FUNCTION_BLOCK F_IS_VALID (* Check if REAL/LREAL is valid (not NaN, not Inf) *)
  (* Standard: 61131-3; Description: Copyright (c) 2013 TU Wien ACIN and others. This program and the accompanying materials are made available under the terms of the Eclipse Public License 2.0 which is available at https://www.eclipse.org/legal/epl-2.0/ SPDX-License-Identifier: EPL-2.0 Some portions generated by Gemini CLI *)
  (* Version 3.1, 2026-01-31, Franz Höpfinger, HR Agrartechnik GmbH, initial API and implementation and/or initial documentation *)
  (* Version 3.0, 2025-04-14, Patrick Aigner, changed package *)
  PACKAGE iec61131::conversion;
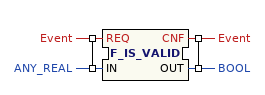
  EVENT_INPUT
    REQ WITH IN; (* Normal Execution Request *)
  END_EVENT
  EVENT_OUTPUT
    CNF WITH OUT; (* Execution Confirmation *)
  END_EVENT
  VAR_INPUT
    IN : ANY_REAL;
  END_VAR
  VAR_OUTPUT
    OUT : BOOL;
  END_VAR
  EC_STATES
    REQ : REQ -> CNF;
  END_STATES
  ALGORITHM REQ IN ST:
OUT := IS_VALID(IN);
  END_ALGORITHM
END_FUNCTION_BLOCK
